Universal Robots PolyScope program: test.urp

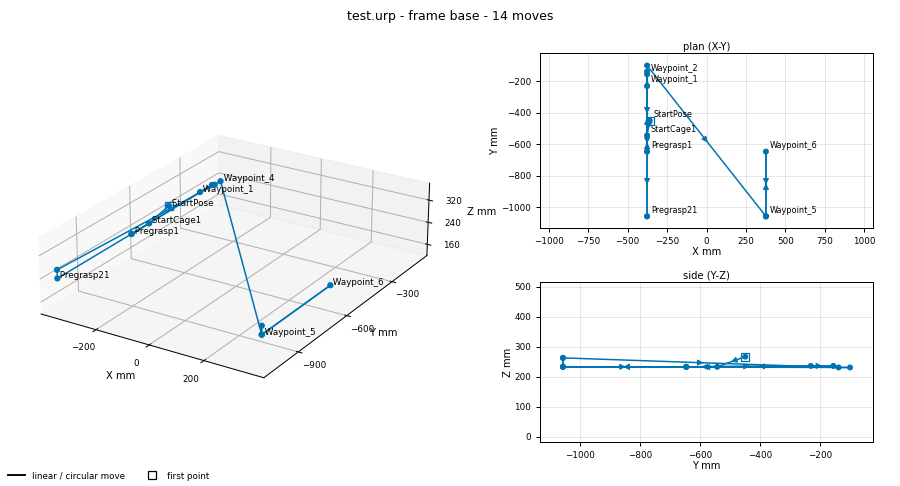
[picture p0: tool path of test.urp in frame base, 14 of 14 moves have a stored position in this frame; points joined in program order, loops and branches not executed]
Program test (installation=default directory=/home/asger/Downloads/ursim-5.11.4.108353/programs/testArla createdIn=5.11.4.108353 lastSavedIn=5.11.4.108353 robotSerialNumber=20195299999)
Calibrated DH parameters: a=[0, -0.6127, -0.57155, 0, 0, 0]; d=[0.1807, 0, 0, 0.17415, 0.11985, 0.11655]; alpha=[1.570796, 0, 0, 1.570796, -1.570796, 0]; deltaTheta=[0, 0, 0, 0, 0, 0]
Robot Program (runOnlyOnce=true)
  Folder ResetForce
    Wait Condition expression=is_steady()
    Wait Sleep waitTime=0.25
    Script: zero_ftsensor()
    Wait Sleep waitTime=0.25
  Timer (action=Start) variable(name=timer_1)
  MoveJ speed 30 deg/s, acceleration 40 deg/s^2 (useActiveTCP=true) feature=Base
    Waypoint StartPose: motionParameters(jointSpeed=0.523599 jointAcceleration=0.698132 cartesianSpeed=0.25 cartesianAcceleration=1.2); TCP in base x=-360.061 y=-449.1 z=267.738 mm, rx=0 ry=3.1416 rz=0 rad; joints [-111.11, -92.71, -132.9, -44.39, 90, -21.11] deg
  Folder Cage1
    MoveL speed 250 mm/s, acceleration 1200 mm/s^2 (useActiveTCP=true) feature=Base
      Waypoint StartCage1: TCP in base x=-377.018 y=-542.594 z=233.918 mm, rx=-0.1647 ry=-3.1372 rz=0.0003 rad; joints [-109.613, -103.066, -125.349, -41.605, 89.828, -13.516] deg
    MoveL speed 250 mm/s, acceleration 1200 mm/s^2 (useActiveTCP=true) feature=Base
      Waypoint Pregrasp1: TCP in base x=-377.023 y=-645.691 z=233.925 mm, rx=0.1472 ry=3.1381 rz=-0.0004 rad; joints [-106.906, -109.721, -115.734, -44.56, 89.809, -11.457] deg
    Force Frame feature=Base; selection=[0, 0, 1, 0, 0, 0]; wrench=[0, 10, 225, 0, 0, 0]; limitsForce=[0.15, 0.15, 0.15, 1.047198, 1.047198, 1.047198]; limitsMotion=[0.1, 0.1, 0.1, 0.349066, 0.349066, 0.349066]
      Set DigitalOutput pin=digital_out[0]; digitalValue=1
      Wait Sleep waitTime=0.5
    MoveL speed 100 mm/s, acceleration 1200 mm/s^2 (useActiveTCP=true) feature=Base
      MoveDirectionNode (selectedDirection=YPlus)
        Until DISTANCE (allowActions=false deceleration=3 distanceNodeType=STOP) Distance=0.1; motionParameters(blendRadius=0)
    Set DigitalOutput pin=digital_out[0]; digitalValue=0
    MoveL speed 250 mm/s, acceleration 1200 mm/s^2 (useActiveTCP=true) feature=Base
      MoveDirectionNode (selectedDirection=YPlus)
        Until DISTANCE (allowActions=false deceleration=3 distanceNodeType=STOP) Distance=0.315; motionParameters(blendRadius=0)
    MoveL speed 250 mm/s, acceleration 1200 mm/s^2 (useActiveTCP=true) feature=Base
      Waypoint Waypoint_1: TCP in base x=-377.05 y=-230.69 z=236.965 mm, rx=-0.1473 ry=-3.1381 rz=-0.0006 rad; joints [-125.334, -81.964, -147.416, -40.639, 89.988, -29.959] deg; TCP offset x=0 y=0 z=0 mm, rx=0 ry=0 rz=0 rad
    MoveL speed 250 mm/s, acceleration 1200 mm/s^2 (useActiveTCP=true) feature=Base
      Waypoint Waypoint_2: TCP in base x=-377.05 y=-155.463 z=236.965 mm, rx=-0.1473 ry=-3.1381 rz=-0.0006 rad; joints [-132.311, -77.472, -150.605, -41.939, 89.986, -36.936] deg
    Wait Sleep waitTime=2
    MoveL speed 250 mm/s, acceleration 1200 mm/s^2 (useActiveTCP=true) feature=Base
      Waypoint Pregrasp1: TCP in base x=-377.023 y=-645.691 z=233.925 mm, rx=0.1472 ry=3.1381 rz=-0.0004 rad; joints [-106.906, -109.721, -115.734, -44.56, 89.809, -11.457] deg
    MoveL speed 250 mm/s, acceleration 1200 mm/s^2 (useActiveTCP=true) feature=Base
      MoveDirectionNode (selectedDirection=ZPlus)
        Until DISTANCE (allowActions=false deceleration=3 distanceNodeType=STOP) Distance=0.005; motionParameters(blendRadius=0)
    MoveL speed 250 mm/s, acceleration 1200 mm/s^2 (useActiveTCP=true) feature=Base
      Waypoint Pregrasp21: TCP in base x=-377.061 y=-1056.7 z=233.886 mm, rx=-0.1648 ry=-3.1372 rz=0.0002 rad; joints [-100.743, -139.405, -64.21, -66.406, 89.701, -4.674] deg
    MoveL speed 300 mm/s, acceleration 1200 mm/s^2 (useActiveTCP=true) feature=Base
      Waypoint Pregrasp22: TCP in base x=-377.043 y=-1056.692 z=263.615 mm, rx=-0.1648 ry=-3.1372 rz=0.0001 rad; joints [-100.742, -138.214, -63.213, -68.601, 89.701, -4.664] deg
    MoveL speed 250 mm/s, acceleration 1200 mm/s^2 (useActiveTCP=true) feature=Base
      MoveDirectionNode (selectedDirection=YPlus)
        Until DISTANCE (allowActions=false deceleration=3 distanceNodeType=STOP) Distance=0.405; motionParameters(blendRadius=0)
    Force Frame feature=Base; selection=[0, 0, 1, 0, 0, 0]; wrench=[0, 10, 225, 0, 0, 0]; limitsForce=[0.15, 0.15, 0.15, 1.047198, 1.047198, 1.047198]; limitsMotion=[0.1, 0.1, 0.1, 0.349066, 0.349066, 0.349066]
      Set DigitalOutput pin=digital_out[0]; digitalValue=1
      Wait Sleep waitTime=0.7
    MoveL speed 250 mm/s, acceleration 1200 mm/s^2 (useActiveTCP=true) feature=Base
      MoveDirectionNode (selectedDirection=YPlus)
        Until DISTANCE (allowActions=false deceleration=3 distanceNodeType=STOP) Distance=0.1; motionParameters(blendRadius=0)
    Set DigitalOutput pin=digital_out[0]; digitalValue=0
    MoveL speed 250 mm/s, acceleration 1200 mm/s^2 (useActiveTCP=true) feature=Base
      MoveDirectionNode (selectedDirection=ZMinus)
        Until DISTANCE (allowActions=false deceleration=3 distanceNodeType=STOP) Distance=0.01; motionParameters(blendRadius=0)
    MoveL speed 250 mm/s, acceleration 1200 mm/s^2 (useActiveTCP=true) feature=Base
      MoveDirectionNode (selectedDirection=YPlus)
        Until DISTANCE (allowActions=false deceleration=3 distanceNodeType=STOP) Distance=0.315; motionParameters(blendRadius=0)
    Halt
    MoveL speed 300 mm/s, acceleration 1200 mm/s^2 (useActiveTCP=true) feature=Base
      Waypoint Waypoint_3: TCP in base x=-376.973 y=-137.77 z=231.649 mm, rx=0.1647 ry=3.1371 rz=0.001 rad; joints [-134.329, -77.453, -151.513, -41.097, 89.885, -38.211] deg
    Halt
    MoveL speed 300 mm/s, acceleration 1200 mm/s^2 (useActiveTCP=true) feature=Base
      Waypoint Waypoint_4: TCP in base x=-376.969 y=-99.845 z=231.657 mm, rx=0.1647 ry=3.1371 rz=0.0009 rad; joints [-138.762, -75.781, -152.558, -41.72, 89.889, -42.641] deg
    Wait Sleep waitTime=2
  Folder Cage2
    MoveL speed 250 mm/s, acceleration 1200 mm/s^2 (useActiveTCP=true) feature=Base
      Waypoint Waypoint_5: TCP in base x=377.06 y=-1056.7 z=233.886 mm, rx=-0.1648 ry=-3.1372 rz=0.0002 rad; joints [-61.432, -139.364, -64.287, -66.345, 89.993, 34.583] deg
    MoveL speed 250 mm/s, acceleration 1200 mm/s^2 (useActiveTCP=true) feature=Base
      Waypoint Waypoint_6: TCP in base x=377.02 y=-645.691 z=233.925 mm, rx=0.1472 ry=3.1381 rz=-0.0004 rad; joints [-46.249, -109.666, -115.769, -44.554, 89.99, 49.121] deg
    Force Frame feature=Base; selection=[0, 0, 1, 0, 0, 0]; wrench=[0, 10, 225, 0, 0, 0]; limitsForce=[0.15, 0.15, 0.15, 1.047198, 1.047198, 1.047198]; limitsMotion=[0.1, 0.1, 0.1, 0.349066, 0.349066, 0.349066]
      Set DigitalOutput pin=digital_out[0]; digitalValue=1
      Wait Sleep waitTime=0.5
    MoveL speed 100 mm/s, acceleration 1200 mm/s^2 (useActiveTCP=true) feature=Base
      MoveDirectionNode (selectedDirection=YPlus)
        Until DISTANCE (allowActions=false deceleration=3 distanceNodeType=STOP) Distance=0.1; motionParameters(blendRadius=0)
    Set DigitalOutput pin=digital_out[0]; digitalValue=0
    MoveL speed 250 mm/s, acceleration 1200 mm/s^2 (useActiveTCP=true) feature=Base
      MoveDirectionNode (selectedDirection=YPlus)
        Until DISTANCE (allowActions=false deceleration=3 distanceNodeType=STOP) Distance=0.315; motionParameters(blendRadius=0)
    Halt
    MoveL speed 250 mm/s, acceleration 1200 mm/s^2 (useActiveTCP=true) feature=Base
      Waypoint Waypoint_5: TCP in base x=377.06 y=-1056.7 z=233.886 mm, rx=-0.1648 ry=-3.1372 rz=0.0002 rad; joints [-61.432, -139.364, -64.287, -66.345, 89.993, 34.583] deg
    MoveL speed 250 mm/s, acceleration 1200 mm/s^2 (useActiveTCP=true) feature=Base
      Waypoint Waypoint_7: TCP in base x=377.04 y=-1056.692 z=263.615 mm, rx=-0.1648 ry=-3.1372 rz=0.0001 rad; joints [-61.433, -138.175, -63.287, -68.537, 89.997, 34.582] deg
    MoveL speed 250 mm/s, acceleration 1200 mm/s^2 (useActiveTCP=true) feature=Base
      MoveDirectionNode (selectedDirection=YPlus)
        Until DISTANCE (allowActions=false deceleration=3 distanceNodeType=STOP) Distance=0.405; motionParameters(blendRadius=0)
    Force Frame feature=Base; selection=[0, 0, 1, 0, 0, 0]; wrench=[0, 10, 225, 0, 0, 0]; limitsForce=[0.15, 0.15, 0.15, 1.047198, 1.047198, 1.047198]; limitsMotion=[0.1, 0.1, 0.1, 0.349066, 0.349066, 0.349066]
      Set DigitalOutput pin=digital_out[0]; digitalValue=1
      Wait Sleep waitTime=0.7
    MoveL speed 250 mm/s, acceleration 1200 mm/s^2 (useActiveTCP=true) feature=Base
      MoveDirectionNode (selectedDirection=YPlus)
        Until DISTANCE (allowActions=false deceleration=3 distanceNodeType=STOP) Distance=0.1; motionParameters(blendRadius=0)
    Set DigitalOutput pin=digital_out[0]; digitalValue=0
    MoveL speed 250 mm/s, acceleration 1200 mm/s^2 (useActiveTCP=true) feature=Base
      MoveDirectionNode (selectedDirection=ZMinus)
        Until DISTANCE (allowActions=false deceleration=3 distanceNodeType=STOP) Distance=0.01; motionParameters(blendRadius=0)
    MoveL speed 250 mm/s, acceleration 1200 mm/s^2 (useActiveTCP=true) feature=Base
      MoveDirectionNode (selectedDirection=YPlus)
        Until DISTANCE (allowActions=false deceleration=3 distanceNodeType=STOP) Distance=0.315; motionParameters(blendRadius=0)
    Halt
  Timer (action=Stop) variable(name=timer_2)
